(* PLC project CoDeSys External Library Template, WAGO e!COCKPIT e!COCKPIT, author 3S - Smart Software Solutions GmbH *)
(* stored: creationDateTime 2019-10-29T12:22:40.3137224, version 3.5.5.30, modificationDateTime 2019-10-24T14:40:07.960949, organization 3S - Smart Software Solutions GmbH *)
(* Library project template with all possible element types, docu and a sample project structure *)

(* values of enumKlasaAlarmu: Bezpieczenstwa: najwyższy priorytet alarmu - alarm mogący mieć wpływ na bezpieczeństwo działania budynku; Krytyczny: wysoki priorytet alarmu - alarm istotny mogący doprowadzić do zaistnienia alarmu bezpieczeństwa; Ostrzezenie: średni priorytet alarmu - ostrzeżenie o nieprawidłowym działaniu któregoś z urządzeń; Informacyjny: niski priorytet alarm wyswietlany nie wymagajacy potwierdzenia; AwariaAutomatyki: alarm (podjrzenia) uszkodzenia lub nieprawidłowego działania automatyki; Wewnetrzny: alarm wewnetrzny niewyświetlany nie wymaga potwierdzenia; Systemowy: alarm systemowy niewyświetlany nie wymaga potwierdzenia *)

(* Nazwa bloku: Enumeracja - definicja klasy błędów Projekt: Bałtyckie Centrum Biznesu Budynek 2 Firma: Solwena Autor: Marcin Szumiło Aktualizacja: 2017-11-17-11:00-PK: aktualizacja względem pliku komunikacja 2019-02-13-14:56-AWy: dodanie klasy AwariaAutomatyki *)
{attribute 'qualified_only'}
{attribute 'strict'}
TYPE enumKlasaAlarmu : (Bezpieczenstwa := 0, Krytyczny := 1, Ostrzezenie := 2, Informacyjny := 3, AwariaAutomatyki := 8, Wewnetrzny := 9, Systemowy := 10);
END_TYPE
